Staubli VAL3: UPLOAD.pgx

public program UpLoad()
  local num l_nKey
  local bool l_bRes
  local num l_nTime
begin
  //不推荐客户自己改动此函数代码
  //-----------------------------------------------------------------------
  //把CS8C的信息上传到上位机中
  cls()
  call UI:Control_PanelMd("正在上传，请等待")
  call UI:Control_BottomS(",,,,,,,终止")
  call TxtFile:CloseFile()
  DataBase:bUpload=true
  l_nTime=clock()


  //开始上传
  while DataBase:bUpload==true and 120-clock()+l_nTime>0
    l_nKey=getKey()

    if l_nKey==278
      call UI:Control_YesNO("确定要终止上传吗",l_bRes)
      if l_bRes
        DataBase:bUpload=false
        return
      else
        call UI:Control_PanelMd("正在上传，请等待")
        call UI:Control_BottomS(",,,,,,,终止")
      endIf
    endIf


    gotoxy(0,12)
    put("剩余:"+toString("",120-clock()+l_nTime)+"秒     ")
    delay(0)

  endWhile

  //对上传结果进行判断
  DataBase:bUpload=false
  if clock()>l_nTime+60
    popUpMsg("上传失败!")
  else
    popUpMsg("上传成功")
  endIf
  cls()

end
